(* Variables for program blocks *)
VAR_GLOBAL PERSISTENT
	
	nPowerFailureCounter					:UINT;
	
END_VAR
VAR_GLOBAL
	
	(* PLC start detected *)
	bFirstCycleDetected						:BOOL;
	bMachineSequenzAktiv					:BOOL;		(* PLC startup done (LED test) program in cyclic mode *)

	(* Clock generator *)
	bClock500ms								:BOOL;		(* Clock 500ms on/off *)
	bClock1s								:BOOL;		(* Clock 1s on/off *)
	bClock2s								:BOOL;		(* Clock 2s on/off *)
	bRisingEdge500ms						:BOOL;		(* Rising edge all 500ms over one cycle *)
	bRisingEdge1s							:BOOL;		(* Edge after 1s over a cycle *)
	bRisingEdge2s							:BOOL;		(* Edge after 2s over a cycle *)

END_VAR
(* End *)

(* stored: Version 1.1.0.1, ProductVersion 3.1.4024.12
   GVL GVL10_VAR_PRG: Id {35ad527e-83a4-4ee6-ae5b-53264e45d32c} *)
